(* IEC 61131-3 sources: Paster/src/fb, 3 files *)

(* ---- FB_ActuatorManager.st ---- *)
FUNCTION_BLOCK FB_ActuatorManager
VAR_INPUT
    // Команды от PasteurManager:
    Pasteur_CircPump_ON     : BOOL;
    Pasteur_Mixer_ON        : BOOL;
    Pasteur_CoolingValve_ON : BOOL;
    Pasteur_HeatPowerReq    : REAL;

    // Команды от CIPManager:
    CIP_Valve_Cold_ON  : BOOL;  // холодная вода (CIP)
    CIP_Valve_Hot_ON   : BOOL;  // горячая вода (CIP)
    CIP_Valve_Alk_ON   : BOOL;
    CIP_Valve_Acid_ON  : BOOL;
    CIP_Pump_ON        : BOOL;
    CIP_DrainValve_ON  : BOOL;
    CIP_Mixer_ON       : BOOL;  // <<< новый вход: мешалка по уставкам этапов CIP

    // Команды от DosingManager:
    Dosing_FillPump_ON : BOOL;

    // Команды от TemperatureManager:
    Temp_DO_Heater1_Cmd : BOOL;
    Temp_DO_Heater2_Cmd : BOOL;
    Temp_DO_Heater3_Cmd : BOOL;
    Temp_AO_HeaterPower : REAL;

    // Mixer/VFD (на будущее):
    VFD_MixerRunReq    : BOOL;
    VFD_MixerRevReq    : BOOL;

    // ===== РУЧНЫЕ КОМАНДЫ (1:1 c физическими DO) =====
    Man1_ValveCold        : BOOL;
    Man2_CircPump         : BOOL;
    Man3_MixerFwd         : BOOL;
    Man4_MixerRev         : BOOL;
    Man5_PumpDisp         : BOOL;
    Man6_Heater1          : BOOL;
    Man7_Heater2          : BOOL;
    Man8_Heater3          : BOOL;
    Man9_ValveCIP_Cold    : BOOL;
    Man10_ValveCIP_Hot    : BOOL;
    Man11_ValveAlk        : BOOL;
    Man12_ValveAcid       : BOOL;
    Man13_PumpCIP         : BOOL;
    Man14_ValveDrain      : BOOL;

    // Флаги режимов:
    Mode_Pasteur_ACTIVE   : BOOL;
    Mode_CIP_ACTIVE       : BOOL;
    Mode_Dosing_ACTIVE    : BOOL;
    Mode_Manual_ACTIVE    : BOOL;
    Mode_Recipe_ACTIVE    : BOOL;

    // Блокировки:
    BLOCK_AllOff          : BOOL;
    BLOCK_HeaterOff       : BOOL;

    // Параметры:
    PAR_UseVFD            : BOOL;
END_VAR

VAR_OUTPUT
    // — Карта выходов ПЛК — (имена строго как в FB_Main)
    DO1_ValveCold       : BOOL; // клапан охлаждения (хол. вода)
    DO2_CircPump        : BOOL; // циркуляционный насос
    DO3_MixerFwd        : BOOL;
    DO4_MixerRev        : BOOL;
    DO5_PumpDisp        : BOOL;
    DO6_Heater1         : BOOL;
    DO7_Heater2         : BOOL;
    DO8_Heater3         : BOOL;
    DO9_ValveCIP_Cold   : BOOL;
    DO10_ValveCIP_Hot   : BOOL;
    DO11_ValveAlk       : BOOL;
    DO12_ValveAcid      : BOOL;
    DO13_PumpCIP        : BOOL;
    DO14_ValveDrain     : BOOL;

    // — Аналог —
    AO_1  : REAL;       // мощность нагрева 0..10 В
    AO_2  : REAL;       // резерв / «старт» (если не VFD)
END_VAR

// ========== Безопасные значения по умолчанию ==========
DO1_ValveCold:=FALSE; DO2_CircPump:=FALSE; DO3_MixerFwd:=FALSE; DO4_MixerRev:=FALSE; DO5_PumpDisp:=FALSE;
DO6_Heater1:=FALSE; DO7_Heater2:=FALSE; DO8_Heater3:=FALSE; DO9_ValveCIP_Cold:=FALSE; DO10_ValveCIP_Hot:=FALSE;
DO11_ValveAlk:=FALSE; DO12_ValveAcid:=FALSE; DO13_PumpCIP:=FALSE; DO14_ValveDrain:=FALSE;
AO_1:=0.0; AO_2:=0.0;

// ========== ЛОГИКА ==========
IF NOT BLOCK_AllOff THEN

    // DO1 — клапан охлаждения (пастеризатор)
    IF Mode_Manual_ACTIVE THEN
        DO1_ValveCold := Man1_ValveCold;
    ELSIF Mode_Pasteur_ACTIVE OR Mode_Recipe_ACTIVE THEN
        DO1_ValveCold := Pasteur_CoolingValve_ON;
    ELSE
        DO1_ValveCold := FALSE;
    END_IF;

    // DO2 — циркуляционный насос (пастеризатор)
    IF Mode_Manual_ACTIVE THEN
        DO2_CircPump := Man2_CircPump;
    ELSIF Mode_CIP_ACTIVE THEN
        DO2_CircPump := FALSE; // при необходимости можно разрешить в CIP
    ELSIF Mode_Pasteur_ACTIVE OR Mode_Recipe_ACTIVE THEN
        DO2_CircPump := Pasteur_CircPump_ON;
    ELSE
        DO2_CircPump := FALSE;
    END_IF;

    // DO3/DO4 — мешалка
    IF Mode_Manual_ACTIVE THEN
        DO3_MixerFwd := Man3_MixerFwd;
        DO4_MixerRev := Man4_MixerRev;
    ELSE
        IF Mode_CIP_ACTIVE THEN
            // В режиме CIP — только вперёд, по сигналу от FB_CIPManager_v2
            DO3_MixerFwd := CIP_Mixer_ON;
            DO4_MixerRev := FALSE;
        ELSIF Mode_Pasteur_ACTIVE OR Mode_Recipe_ACTIVE THEN
            DO3_MixerFwd := Pasteur_Mixer_ON;
            DO4_MixerRev := FALSE;
        ELSE
            DO3_MixerFwd := FALSE;
            DO4_MixerRev := FALSE;
        END_IF;
    END_IF;

    // защита от одновременного FWD/REV
    IF DO3_MixerFwd AND DO4_MixerRev THEN
        DO4_MixerRev := FALSE;
    END_IF;

    // DO5 — насос розлива/дозирования
    IF Mode_Manual_ACTIVE THEN
        DO5_PumpDisp := Man5_PumpDisp;
    ELSIF Mode_Dosing_ACTIVE THEN
        DO5_PumpDisp := Dosing_FillPump_ON;
    ELSE
        DO5_PumpDisp := FALSE;
    END_IF;

    // DO6..DO8 — нагрев и AO_1
    IF BLOCK_HeaterOff THEN
        DO6_Heater1 := FALSE; DO7_Heater2 := FALSE; DO8_Heater3 := FALSE;
        AO_1 := 0.0;
    ELSIF Mode_Manual_ACTIVE THEN
        DO6_Heater1 := Man6_Heater1;
        DO7_Heater2 := Man7_Heater2;
        DO8_Heater3 := Man8_Heater3;
        AO_1 := 0.0;
    ELSE
        DO6_Heater1 := Temp_DO_Heater1_Cmd;
        DO7_Heater2 := Temp_DO_Heater2_Cmd;
        DO8_Heater3 := Temp_DO_Heater3_Cmd;
        AO_1 := Temp_AO_HeaterPower;
    END_IF;

    // DO9..DO14 — CIP-исполнительные механизмы
    IF Mode_Manual_ACTIVE THEN
        DO9_ValveCIP_Cold := Man9_ValveCIP_Cold;
    ELSIF Mode_CIP_ACTIVE THEN
        DO9_ValveCIP_Cold := CIP_Valve_Cold_ON;
    ELSE
        DO9_ValveCIP_Cold := FALSE;
    END_IF;

    IF Mode_Manual_ACTIVE THEN
        DO10_ValveCIP_Hot := Man10_ValveCIP_Hot;
    ELSIF Mode_CIP_ACTIVE THEN
        DO10_ValveCIP_Hot := CIP_Valve_Hot_ON;
    ELSE
        DO10_ValveCIP_Hot := FALSE;
    END_IF;

    IF Mode_Manual_ACTIVE THEN
        DO11_ValveAlk := Man11_ValveAlk;
    ELSIF Mode_CIP_ACTIVE THEN
        DO11_ValveAlk := CIP_Valve_Alk_ON;
    ELSE
        DO11_ValveAlk := FALSE;
    END_IF;

    IF Mode_Manual_ACTIVE THEN
        DO12_ValveAcid := Man12_ValveAcid;
    ELSIF Mode_CIP_ACTIVE THEN
        DO12_ValveAcid := CIP_Valve_Acid_ON;
    ELSE
        DO12_ValveAcid := FALSE;
    END_IF;

    IF Mode_Manual_ACTIVE THEN
        DO13_PumpCIP := Man13_PumpCIP;
    ELSIF Mode_CIP_ACTIVE THEN
        DO13_PumpCIP := CIP_Pump_ON;
    ELSE
        DO13_PumpCIP := FALSE;
    END_IF;

    IF Mode_Manual_ACTIVE THEN
        DO14_ValveDrain := Man14_ValveDrain;
    ELSIF Mode_CIP_ACTIVE THEN
        DO14_ValveDrain := CIP_DrainValve_ON;
    ELSE
        DO14_ValveDrain := FALSE;
    END_IF;

    // AO_2 — если VFD не используется (имитация «старта»)
    IF NOT PAR_UseVFD THEN
        IF DO3_MixerFwd OR DO4_MixerRev THEN
            AO_2 := 100.0; // %
        ELSE
            AO_2 := 0.0;
        END_IF;
    ELSE
        AO_2 := 0.0;
    END_IF;

END_IF;

END_FUNCTION_BLOCK

(* ---- FB_DosingManager.st ---- *)
FUNCTION_BLOCK FB_DosingManager
VAR_INPUT
    EN_Continuous        : BOOL;  // запрос непрерывного розлива (уровень)
    EN_Portion           : BOOL;  // запрос дозированного розлива (уровень)

    PAR_UseGunSensor     : BOOL;  // ждать сигнал "пистолет на месте"
    GunSensor            : BOOL;  // TRUE = пистолет на месте

    PAR_UsePortionButton : BOOL;  // использовать внешнюю кнопку порции
    PortionButton        : BOOL;  // TRUE = кнопка нажата

    SP_DoseVolume        : REAL;  // объём дозы, л
    FlowMeter            : REAL;  // ОБЩИЙ/АБСОЛЮТНЫЙ накопленный объём, л (счётчик)
END_VAR

VAR_OUTPUT
    FillPump_ON  : BOOL;  // команда на насос розлива (DO5)
    PortionDone  : BOOL;  // завершение дозы (импульсом)
END_VAR

VAR
    dosingActive      : BOOL := FALSE;  // в процессе дозирования
    flowBaseAtStart   : REAL := 0.0;    // база счётчика на старте дозы
    doseAccum         : REAL := 0.0;    // дельта объёма с начала дозы
    init_done         : BOOL := FALSE;
    canStart          : BOOL := FALSE;
END_VAR

// --- одноразовая инициализация ---
IF NOT init_done THEN
    FillPump_ON := FALSE;
    PortionDone := FALSE;
    dosingActive := FALSE;
    flowBaseAtStart := 0.0;
    doseAccum := 0.0;
    init_done := TRUE;
END_IF;

// сбрасываем "готово" по умолчанию (если нужна защёлка — реализовать снаружи)
PortionDone := FALSE;

// ===== ПОРЦИОННЫЙ РЕЖИМ (имеет приоритет над непрерывным) =====
IF EN_Portion THEN

    IF NOT dosingActive THEN
        // проверяем условия старта
        canStart := TRUE;

        IF PAR_UsePortionButton THEN
            canStart := canStart AND PortionButton;
        END_IF;

        IF PAR_UseGunSensor THEN
            canStart := canStart AND GunSensor;
        END_IF;

        IF canStart THEN
            dosingActive := TRUE;
            flowBaseAtStart := FlowMeter;   // запоминаем базу абсолютного счётчика
            doseAccum := 0.0;
            FillPump_ON := TRUE;
        ELSE
            FillPump_ON := FALSE;
        END_IF;

    ELSE
        // доза идёт
        doseAccum := FlowMeter - flowBaseAtStart;
        IF doseAccum < 0.0 THEN
            // защита от возможного переполнения/обнуления счётчика
            flowBaseAtStart := FlowMeter;
            doseAccum := 0.0;
        END_IF;

        IF doseAccum >= SP_DoseVolume THEN
            // доза набрана — корректная остановка, флаг завершения
            FillPump_ON := FALSE;
            PortionDone := TRUE;
            dosingActive := FALSE;
            doseAccum := 0.0;

        ELSE
            // при снятом пистолете — пауза насоса, но дозирование не сбрасываем
            IF PAR_UseGunSensor AND (NOT GunSensor) THEN
                FillPump_ON := FALSE;
            ELSE
                FillPump_ON := TRUE;
            END_IF;
        END_IF;
    END_IF;

ELSE
    // порционный режим выключен — аварийный/принудительный выход из дозы
    dosingActive := FALSE;
    doseAccum := 0.0;
END_IF;

// ===== НЕПРЕРЫВНЫЙ РЕЖИМ (работает, только когда порционный не активен) =====
IF (NOT EN_Portion) AND (NOT dosingActive) THEN
    IF EN_Continuous THEN
        IF PAR_UseGunSensor THEN
            FillPump_ON := GunSensor;   // только при "пистолет на месте"
        ELSE
            FillPump_ON := TRUE;
        END_IF;
    ELSE
        FillPump_ON := FALSE;
    END_IF;
END_IF;

END_FUNCTION_BLOCK

(* ---- FB_SoftFlowmeter.st ---- *)
FUNCTION_BLOCK FB_SoftFlowmeter
VAR_INPUT
    Enable     : BOOL;   // разрешение интегратора
    Seconds_UD : UDINT;  // секундный тик (монотонный)
    PumpOn     : BOOL;   // насос работает
    Rate_Lps   : REAL;   // производительность, л/с
    Reset      : BOOL;   // сброс накопления
END_VAR

VAR_OUTPUT
    FlowAbs_L  : REAL;   // накопленный объём, л (абсолют)
    Delta_L    : REAL;   // прирост за последний шаг, л
END_VAR

VAR
    init_done  : BOOL  := FALSE;
    lastSec_UD : UDINT := 0;
    accum_L    : REAL  := 0.0;
    secDiff_UD : UDINT := 0;    // <-- выносим сюда
END_VAR

// --- инициализация ---
IF NOT init_done THEN
    lastSec_UD := Seconds_UD;
    accum_L    := 0.0;
    FlowAbs_L  := 0.0;
    Delta_L    := 0.0;
    init_done  := TRUE;
END_IF;

// --- сброс ---
IF Reset THEN
    accum_L   := 0.0;
    FlowAbs_L := 0.0;
    Delta_L   := 0.0;
END_IF;

// --- по умолчанию прирост = 0 ---
Delta_L := 0.0;

// --- основной цикл интеграции ---
IF Enable THEN
    IF Seconds_UD <> lastSec_UD THEN
        secDiff_UD := Seconds_UD - lastSec_UD;
        IF secDiff_UD > 10 THEN secDiff_UD := 10; END_IF;   // защита от «рывка»
        lastSec_UD := Seconds_UD;

        IF PumpOn THEN
            Delta_L := Rate_Lps * UDINT_TO_REAL(secDiff_UD); // правильное приведение
            IF Delta_L < 0.0 THEN Delta_L := 0.0; END_IF;
            accum_L := accum_L + Delta_L;
        END_IF;
    END_IF;
END_IF;

// защита от отрицательных
IF accum_L < 0.0 THEN accum_L := 0.0; END_IF;
FlowAbs_L := accum_L;

END_FUNCTION_BLOCK
